// TIA Portal V17 export
// export: Created 2025-05-06T14:34:18.18359Z, ExportSetting WithDefaults, DisplayName Totally Integrated Automation Portal, DisplayVersion V17 Update 8, DisplayName TIA Portal Openness, DisplayVersion V17 Update 8, DisplayName TIA Portal Version Control Interface, DisplayVersion V17, DisplayName SINAMICS Startdrive Advanced, DisplayVersion V17 SP2, DisplayName SINAMICS Startdrive G110M, G120, G120C, G120D, G120P, G115D, DisplayVersion V17 SP2, DisplayName SINAMICS Startdrive G130, G150, S120, S150, SINAMICS MV, S210, DisplayVersion V17 SP2, DisplayName STEP 7 Professional, DisplayVersion V17 Update 8, DisplayName SINUMERIK ONE STEP 7 Toolbox, DisplayVersion V17 Update 12, DisplayName SINUMERIK 840D sl STEP 7 Toolbox, DisplayVersion V17 Update 12, DisplayName STEP 7 Safety, DisplayVersion V17 Update 6, DisplayName WinCC Advanced, DisplayVersion V17 Update 8
DATA_BLOCK "DB16100_OPC_UA_MAINTENANCE_HMI"   // DB16100
{ S7_Optimized_Access := 'FALSE'; DB_Accessible_From_OPC_UA := 'FALSE' }
VERSION : 0.1
// stored: AutoNumber false, DBAccessibleFromOPCUA false, DBAccessibleFromWebserver true, IsOnlyStoredInLoadMemory false, IsWriteProtectedInAS false
   VAR
      HMI_BUTTON : Struct
         ACKNOWLEDGE_ACTION_BUTTON : Bool;
         SPARE_1 : Bool;
         SPARE_2 : Bool;
         SPARE_3 : Bool;
         SPARE_4 : Bool;
         SPARE_5 : Bool;
         SPARE_6 : Bool;
         SPARE_7 : Bool;
         SPARE_8 : Bool;
         SPARE_9 : Bool;
         SPARE_10 : Bool;
         SPARE_11 : Bool;
         SPARE_12 : Bool;
         SPARE_13 : Bool;
         SPARE_14 : Bool;
         SPARE_15 : Bool;
      END_STRUCT;
      MAINTENANCE_ACTION_LIST_VALUE : Int;
      MAINTENANCE_HMI_VALUE_1 : Int;
      MAINTENANCE_HMI_VALUE_2 : Int;
      MAINTENANCE_HMI_VALUE_3 : Int;
      MAINTENANCE_HMI_VALUE_4 : Int;
      MAINTENANCE_HMI_VALUE_5 : Int;
      MAINTENANCE_HMI_VALUE_6 : Int;
      MAINTENANCE_HMI_VALUE_7 : Int;
      MAINTENANCE_HMI_VALUE_8 : Int;
      MAINTENANCE_HMI_VALUE_9 : Int;
      MAINTENANCE_HMI_VALUE_10 : Int;
      MAINTENANCE_HMI_VALUE_11 : Int;
      MAINTENANCE_HMI_VALUE_12 : Int;
      MAINTENANCE_HMI_BIT_VALUE_1 : Bool;
   END_VAR
BEGIN
END_DATA_BLOCK
